FUNCTION_BLOCK LinkFactory IMPLEMENTS I_LinkFactory

METHOD PUBLIC Create : I_Link
VAR_INPUT
	LinkId : T_MAXSTRING;
	LinkSourceNode : I_Node;
	LinkSourcePortName : STRING;
	LinkDestinationNode : I_Node;
	LinkDestinationPortName : STRING;
END_VAR
VAR
	source : I_HaveOutputPorts;
	destination : I_HaveInputPorts;
	pointerToLink : POINTER TO Link;
END_VAR
IF NOT __QUERYINTERFACE(LinkSourceNode,source) THEN
	RETURN;
END_IF

IF NOT __QUERYINTERFACE(LinkDestinationNode,destination) THEN
	RETURN;
END_IF

pointerToLink := __NEW(
	Link(
		Id := LinkId,
		SourceNode := source,
		SourcePortName := LinkSourcePortName,
		DestinationNode := destination,
		DestinationPortName := LinkDestinationPortName
	)
);
Create := pointerToLink^;
END_METHOD

END_FUNCTION_BLOCK

(* stored: Version 1.1.0.1, ProductVersion 3.1.4024.12
   POU LinkFactory: Id {b726a403-2d2b-01c8-3bad-4af7f3f37d51}, SpecialFunc None
   Method Create: Id {f455afd1-37a3-0d6f-23a4-94724961c8cc} *)
